(* CoDeSys 2.3.10.0 project: ServoDistance.pro *)
(* Libraries: STANDARD.LIB 5.6.98 12:03:02 *)

(* Task configuration *)
TASK Standard (PRIORITY := 0, INTERVAL := T#10ms);
	MAIN();
END_TASK

(* Global variable list: Global_Variables *)
VAR_GLOBAL
	Zielona_1 		AT 	%Q* 	:	 BOOL:= 0;
	Zielona_2 		AT 	%Q* 	:	 BOOL:= 0;
	Zielona_3 		AT 	%Q* 	:	 BOOL:= 0;
	Zielona_4 		AT 	%Q* 	:	 BOOL:= 0;

	Czerwona_1 		AT 	%Q*		:	 BOOL:= 0;
	Czerwona_2 		AT 	%Q*		:	 BOOL:= 0;
	Czerwona_3 		AT	%Q*		:	 BOOL:= 0;
	Czerwona_4 		AT 	%Q*		:	 BOOL:= 0;

	Przycisk_1 		AT 	%I*		:	BOOL;
	Przycisk_2 		AT 	%I*		: 	BOOL;
	Przycisk_3 		AT 	%I*		: 	BOOL;
	Przycisk_4 		AT 	%I*		: 	BOOL;

	Scale_1			AT	%Q*		:	INT;
	Scale_2			AT	%Q*		:	INT;

	Enable_1		AT	%Q*		:	BOOL;
	Enable_2		AT 	%Q*		:	BOOL;

	axis1_Not_moving		AT 	%I*		:	BOOL;
	axis1_Moving_Fv		AT 	%I*		:	BOOL;
	axis1_Moving_Bw		AT 	%I*		:	BOOL;
	axis1_position		AT 	%I*		:	LREAL;
	axis1_velo		AT 	%I*		:	LREAL;
	axis1_override		AT 	%Q*		:	UDINT;
	axis1_driving_time		AT 	%Q*		:	TIME;

	axis2_Not_moving		AT 	%I*		:	BOOL;
	axis2_Moving_Fv		AT 	%I*		:	BOOL;
	axis2_Moving_Bw		AT 	%I*		:	BOOL;
	axis2_position		AT 	%I*		:	LREAL;
	axis2_velo		AT 	%I*		:	LREAL;
	axis2_override		AT 	%Q*		:	UDINT;
	axis2_driving_time		AT 	%Q*		:	TIME;
END_VAR

(* Global variable list: TwinCAT_Configuration *)
(* Generated automatically by TwinCAT - (read only) *)
VAR_CONFIG
	.Zielona_1 AT %QX0.0 : BOOL;	(*  ~ {LinkedWith:TIID^Device 2 (EtherCAT (v2.10 only))^Term 1 (CX1100-0004)^Term 5 (EL2004)^Channel 1^Output} *)
	.Zielona_2 AT %QX0.1 : BOOL;	(*  ~ {LinkedWith:TIID^Device 2 (EtherCAT (v2.10 only))^Term 1 (CX1100-0004)^Term 5 (EL2004)^Channel 2^Output} *)
	.Zielona_3 AT %QX0.2 : BOOL;	(*  ~ {LinkedWith:TIID^Device 2 (EtherCAT (v2.10 only))^Term 8 (EK1100)^Term 12 (EL2004)^Channel 1^Output} *)
	.Zielona_4 AT %QX0.3 : BOOL;	(*  ~ {LinkedWith:TIID^Device 2 (EtherCAT (v2.10 only))^Term 8 (EK1100)^Term 12 (EL2004)^Channel 2^Output} *)
	.Czerwona_1 AT %QX0.4 : BOOL;	(*  ~ {LinkedWith:TIID^Device 2 (EtherCAT (v2.10 only))^Term 1 (CX1100-0004)^Term 4 (EL2004)^Channel 1^Output} *)
	.Czerwona_2 AT %QX0.5 : BOOL;	(*  ~ {LinkedWith:TIID^Device 2 (EtherCAT (v2.10 only))^Term 1 (CX1100-0004)^Term 4 (EL2004)^Channel 2^Output} *)
	.Czerwona_3 AT %QX0.6 : BOOL;	(*  ~ {LinkedWith:TIID^Device 2 (EtherCAT (v2.10 only))^Term 8 (EK1100)^Term 11 (EL2004)^Channel 1^Output} *)
	.Czerwona_4 AT %QX0.7 : BOOL;	(*  ~ {LinkedWith:TIID^Device 2 (EtherCAT (v2.10 only))^Term 8 (EK1100)^Term 11 (EL2004)^Channel 2^Output} *)
	.Przycisk_1 AT %IX0.0 : BOOL;
	.Przycisk_2 AT %IX0.1 : BOOL;
	.Przycisk_3 AT %IX0.2 : BOOL;
	.Przycisk_4 AT %IX0.3 : BOOL;
	.Scale_1 AT %QB12 : INT;
	.Scale_2 AT %QB14 : INT;
	.Enable_1 AT %QX16.0 : BOOL;	(*  ~ {LinkedWith:TINC^NC-Task 1 SAF^Axes^Axis 6^Inputs^Axis 6_FromPlc^ControlDWord^Enable;TINC^NC-Task 1 SAF^Axes^Axis 6^Inputs^Axis 6_FromPlc^ControlDWord^FeedEnablePlus;TINC^NC-Task 1 SAF^Axes^Axis 6^Inputs^Axis 6_FromPlc^ControlDWord^FeedEnableMinus} *)
	.Enable_2 AT %QX16.1 : BOOL;	(*  ~ {LinkedWith:TINC^NC-Task 1 SAF^Axes^Axis 8^Inputs^Axis 8_FromPlc^ControlDWord^Enable;TINC^NC-Task 1 SAF^Axes^Axis 8^Inputs^Axis 8_FromPlc^ControlDWord^FeedEnablePlus;TINC^NC-Task 1 SAF^Axes^Axis 8^Inputs^Axis 8_FromPlc^ControlDWord^FeedEnableMinus} *)
	.axis1_Not_moving AT %IX8.0 : BOOL;	(*  ~ {LinkedWith:TINC^NC-Task 1 SAF^Axes^Axis 6^Outputs^Axis 6_ToPlc^StateDWord^NotMoving} *)
	.axis1_Moving_Fv AT %IX8.1 : BOOL;	(*  ~ {LinkedWith:TINC^NC-Task 1 SAF^Axes^Axis 6^Outputs^Axis 6_ToPlc^StateDWord^PositiveDirection} *)
	.axis1_Moving_Bw AT %IX8.2 : BOOL;	(*  ~ {LinkedWith:TINC^NC-Task 1 SAF^Axes^Axis 6^Outputs^Axis 6_ToPlc^StateDWord^NegativeDirection} *)
	.axis1_position AT %IB44 : LREAL;	(*  ~ {LinkedWith:TINC^NC-Task 1 SAF^Axes^Axis 6^Outputs^Axis 6_ToPlc^ActPos} *)
	.axis1_velo AT %IB52 : LREAL;	(*  ~ {LinkedWith:TINC^NC-Task 1 SAF^Axes^Axis 6^Outputs^Axis 6_ToPlc^ActVelo} *)
	.axis1_override AT %QB28 : UDINT;	(*  ~ {LinkedWith:TINC^NC-Task 1 SAF^Axes^Axis 6^Inputs^Axis 6_FromPlc^Override} *)
	.axis1_driving_time AT %QB20 : TIME;
	.axis2_Not_moving AT %IX8.3 : BOOL;	(*  ~ {LinkedWith:TINC^NC-Task 1 SAF^Axes^Axis 8^Outputs^Axis 8_ToPlc^StateDWord^NotMoving} *)
	.axis2_Moving_Fv AT %IX8.4 : BOOL;	(*  ~ {LinkedWith:TINC^NC-Task 1 SAF^Axes^Axis 8^Outputs^Axis 8_ToPlc^StateDWord^PositiveDirection} *)
	.axis2_Moving_Bw AT %IX8.5 : BOOL;	(*  ~ {LinkedWith:TINC^NC-Task 1 SAF^Axes^Axis 8^Outputs^Axis 8_ToPlc^StateDWord^NegativeDirection} *)
	.axis2_position AT %IB34 : LREAL;	(*  ~ {LinkedWith:TINC^NC-Task 1 SAF^Axes^Axis 8^Outputs^Axis 8_ToPlc^ActPos} *)
	.axis2_velo AT %IB60 : LREAL;	(*  ~ {LinkedWith:TINC^NC-Task 1 SAF^Axes^Axis 8^Outputs^Axis 8_ToPlc^ActVelo} *)
	.axis2_override AT %QB32 : UDINT;	(*  ~ {LinkedWith:TINC^NC-Task 1 SAF^Axes^Axis 8^Inputs^Axis 8_FromPlc^Override} *)
	.axis2_driving_time AT %QB24 : TIME;
END_VAR

(* POU MAIN, ST *)
PROGRAM MAIN
VAR
	stoper_axis1: STOPWATCH := (max_value:=t#600s);
	stoper_axis2: STOPWATCH := (max_value:=t#600s);
END_VAR
Czerwona_1 :=  NOT Przycisk_1;
Czerwona_2 :=  NOT Przycisk_2;
Czerwona_3 :=  NOT Przycisk_3;
Czerwona_4 :=  NOT Przycisk_4;

Zielona_1:=  Przycisk_1;
Zielona_2:=  Przycisk_2;
Zielona_3:=  Przycisk_3;
Zielona_4:=  Przycisk_4;

Enable_1 := NOT stoper_axis1.timer.Q;
Enable_2 := NOT stoper_axis2.timer.Q;

Scale_1 := 100;
axis1_override:= 100 * 10000;
Scale_2 := 100;
axis2_override:= 100 * 10000;

stoper_axis1.start_stop := NOT axis1_Not_moving;
stoper_axis1();
axis1_driving_time := stoper_axis1.value;
stoper_axis2.start_stop := NOT axis2_Not_moving;
stoper_axis2();
axis2_driving_time := stoper_axis2.value;
END_PROGRAM

(* POU STOPWATCH, ST *)
FUNCTION_BLOCK STOPWATCH
VAR_INPUT
	max_value: TIME:=t#10S;
	start_stop: BOOL := FALSE;
END_VAR
VAR_OUTPUT
	value: TIME := t#0s;
END_VAR
VAR
	timer: TON;
END_VAR
IF timer.PT <> max_value THEN
	timer.PT := max_value;
END_IF;

IF start_stop = TRUE THEN
	timer(IN:=TRUE);
	value :=timer.ET;
ELSE
	IF timer.IN THEN
		value :=timer.ET;
	END_IF;
	timer(IN:=FALSE);
END_IF;
END_FUNCTION_BLOCK

(* Visualisation StandState
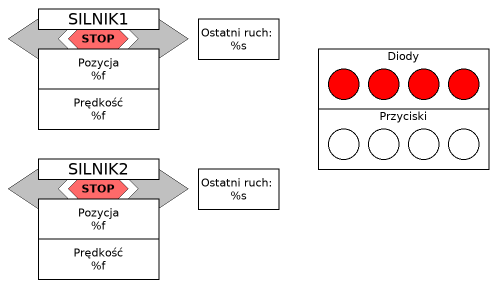
rounded rectangle at (340,110)-(511,171): text "Diody"
polygon at (150,80)-(210,120): invisible if NOT axis1_Moving_Fv
polygon at (30,80)-(90,120): invisible if NOT axis1_Moving_Bw
polygon at (90,90)-(150,110): text "STOP"; invisible if NOT axis1_Not_moving
ellipse at (350,130)-(381,161): invisible if NOT Zielona_1
polygon at (150,230)-(210,270): invisible if NOT axis2_Moving_Fv
polygon at (30,230)-(90,270): invisible if NOT axis2_Moving_Bw
polygon at (90,240)-(150,260): text "STOP"; invisible if NOT axis2_Not_moving
ellipse at (350,130)-(381,161): invisible if NOT Czerwona_1
rectangle at (220,80)-(301,121): text "Ostatni ruch: / %s"; shows MAIN.stoper_axis1.value
rectangle at (220,230)-(301,271): text "Ostatni ruch: / %s"; shows MAIN.stoper_axis2.value
ellipse at (390,130)-(421,161): invisible if NOT Zielona_2
ellipse at (390,130)-(421,161): invisible if NOT Czerwona_2
ellipse at (430,130)-(461,161): invisible if NOT Zielona_3
ellipse at (430,130)-(461,161): invisible if NOT Czerwona_3
ellipse at (470,130)-(501,161): invisible if NOT Zielona_4
ellipse at (470,130)-(501,161): invisible if NOT Czerwona_4
rectangle at (60,70)-(181,91): text "SILNIK1"
rectangle at (60,220)-(181,241): text "SILNIK2"
rounded rectangle at (340,170)-(511,231): text "Przyciski"
ellipse at (350,190)-(381,221): alarm colour if Przycisk_1
ellipse at (390,190)-(421,221): alarm colour if Przycisk_2
ellipse at (430,190)-(461,221): alarm colour if Przycisk_3
ellipse at (470,190)-(501,221): alarm colour if Przycisk_4
rectangle at (60,110)-(181,151): text "Pozycja / %f"; shows axis1_position
rectangle at (60,260)-(181,301): text "Pozycja / %f"; shows axis2_position
rectangle at (60,150)-(181,191): text "Prędkość / %f"; shows axis1_velo
rectangle at (60,300)-(181,341): text "Prędkość / %f"; shows axis2_velo
*)
